PROGRAM MAIN
VAR
	DI2 AT %I*: USINT;
	DI1 AT %I*: USINT;
END_VAR
VAR_OUTPUT
	OUTDI2: USINT;
	OUTDI1: USINT;
END_VAR
VAR
	Count AT %I*: REAL;
END_VAR
VAR_OUTPUT
	Count_Out: REAL;
END_VAR

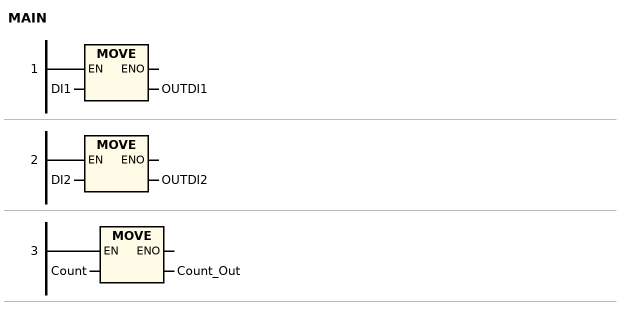
// NETWORK 1
OUTDI1 := DI1;

// NETWORK 2
OUTDI2 := DI2;

// NETWORK 3
Count_Out := Count;

END_PROGRAM

(* stored: Version 1.1.0.1, ProductVersion 3.1.4024.3
   POU MAIN: Id {0393bd89-db80-46d8-b095-12fbe1d1f09e}, SpecialFunc None *)
